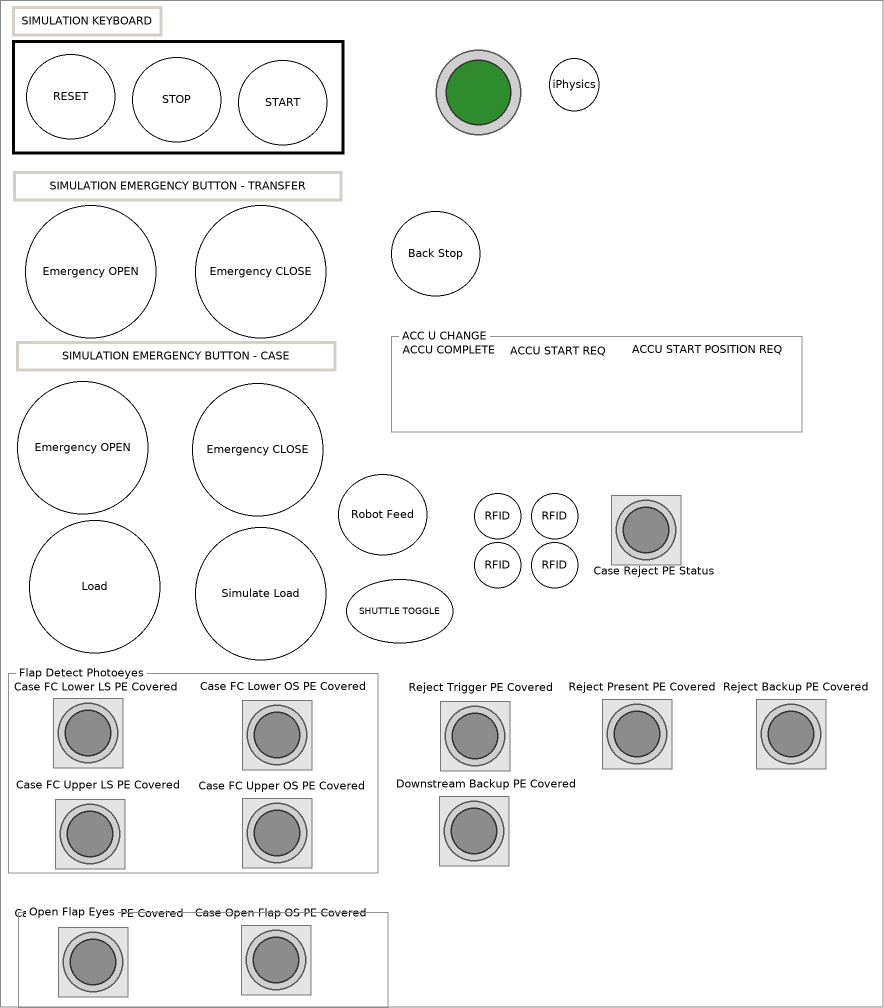
VISUALIZATION Casepacker_Keyboard  // 884x1008
    Rectangle (12,40 332x114)
    Ellipse (26,54 89x85), "RESET"
        tap csp_transfer_main_services_pushbuttons.visu_reset
    Ellipse (132,57 89x85), "STOP"
        tap csp_transfer_main_services_pushbuttons.visu_stop
    Ellipse (238,60 89x85), "START"
        tap csp_transfer_main_services_pushbuttons.visu_start
    Textfield (12,6 150x30), "SIMULATION KEYBOARD"
    Ellipse (25,205 131x133), "Emergency OPEN"
        tap csp_transfer_main_services_pushbuttons.visu_emergency_open
    Ellipse (195,205 131x133), "Emergency CLOSE"
        tap csp_transfer_main_services_pushbuttons.visu_emergency_close
    Textfield (13,171 329x30), "SIMULATION EMERGENCY BUTTON - TRANSFER"
    Lamp1 (426,43 105x99), variable: csp_transfer_main_safety_emergency.HMI_button_lamp_do.field.status, style: Lamp-Lamp1-Green
    Ellipse (391,211 89x85), "Back Stop", colour toggle: csp_transfer_upstacker_sensors.debug_carton_backstop
        toggle csp_transfer_upstacker_sensors.debug_carton_backstop
    Ellipse (192,383 131x133), "Emergency CLOSE"
        tap csp_case_main_services_pushbuttons.visu_emergency_close
    Textfield (16,341 320x30), "SIMULATION EMERGENCY BUTTON - CASE"
    Ellipse (17,381 131x133), "Emergency OPEN"
        tap csp_case_main_services_pushbuttons.visu_emergency_open
    Ellipse (549,58 50x53), "iPhysics"
        toggle MAIN.IP_enable
    GroupBox (8,665 370x208), "Flap Detect Photoeyes"
        PushSwitchLed (45,33 70x70), variable: dbg_csp_case_fc_ls_lower_sensors.flap_chksect_shd.force_input_status, behaviour: TOGGLE, style: Switch-PushSwitchLed-Gray
    Ellipse (29,520 131x133), "Load"
        tap csp_case_loader.load_request
    Ellipse (531,493 47x46), "RFID"
        toggle csp_case_closing_ls_upper.rfid_fake
    Ellipse (531,542 47x46), "RFID"
        toggle csp_case_closing_ls_lower.rfid_fake
    Ellipse (474,493 47x46), "RFID"
        toggle csp_case_closing_os_upper.rfid_fake
    Ellipse (474,542 47x46), "RFID"
        toggle csp_case_closing_os_lower.rfid_fake
    PushSwitchLed (611,495 70x70), behaviour: TOGGLE, style: Switch-PushSwitchLed-Gray
    Label (579,556 150x30), "Case Reject PE Status"
    Ellipse (195,527 131x133), "Simulate Load"
        tap csp_case_transport.product_loaded
    Label (8,673 176x28), "Case FC Lower LS PE Covered"
    PushSwitchLed (55,799 70x70), variable: dbg_csp_case_fc_ls_upper_sensors.flap_chksect_shd.force_input_status, behaviour: TOGGLE, style: Switch-PushSwitchLed-Gray
    Label (10,775 176x20), "Case FC Upper LS PE Covered"
    PushSwitchLed (242,700 70x70), variable: dbg_csp_case_fc_os_lower_sensors.flap_chksect_shd.force_input_status, behaviour: TOGGLE, style: Switch-PushSwitchLed-Gray
    Label (195,678 176x17), "Case FC Lower OS PE Covered"
    PushSwitchLed (242,798 70x70), variable: dbg_csp_case_fc_os_upper_sensors.flap_chksect_shd.force_input_status, behaviour: TOGGLE, style: Switch-PushSwitchLed-Gray
    Label (194,777 176x18), "Case FC Upper OS PE Covered"
    Label (8,888 176x28)
    PushSwitchLed (58,927 70x70), variable: dbg_csp_case_openflap_sensors.open_flap_ls_di_dchk_shd.force_input_status, behaviour: TOGGLE, style: Switch-PushSwitchLed-Gray
    Label (11,905 176x17), "Case Open Flap LS PE Covered"
    PushSwitchLed (241,925 70x70), variable: dbg_csp_case_openflap_sensors.open_flap_os_di_dchk_shd.force_input_status, behaviour: TOGGLE, style: Switch-PushSwitchLed-Gray
    Label (193,904 176x18), "Case Open Flap OS PE Covered"
    GroupBox (391,328 411x104), "ACC U CHANGE"
        Label (381,-232 176x28)
        Label (79,9 176x28), "ACCU START REQ"
    PushSwitchLed (440,701 70x70), variable: dbg_csp_case_discharge_reject_sensors.reject_trigger_inchoerence_chksect_shd.force_input_status, behaviour: TOGGLE, style: Switch-PushSwitchLed-Gray
    Label (393,679 176x17), "Reject Trigger PE Covered"
    PushSwitchLed (602,699 70x70), variable: dbg_csp_case_discharge_reject_sensors.reject_present_di_shd.is_covered, behaviour: TOGGLE, style: Switch-PushSwitchLed-Gray
    Label (554,678 176x18), "Reject Present PE Covered"
    PushSwitchLed (756,699 70x70), variable: dbg_csp_case_discharge_reject_sensors.reject_backup_di_shd.is_covered, behaviour: TOGGLE, style: Switch-PushSwitchLed-Gray
    Label (708,678 176x18), "Reject Backup PE Covered"
    PushSwitchLed (439,796 70x70), variable: dbg_csp_case_discharge_reject_sensors.downstream_backup_di_shd.is_covered, behaviour: TOGGLE, style: Switch-PushSwitchLed-Gray
    Label (391,775 190x18), "Downstream Backup PE Covered"
    Ellipse (338,474 89x81), "Robot Feed"
        toggle csp_case_feed.Feed_request
    Ellipse (346,579 107x64), "SHUTTLE TOGGLE"
        toggle csp_case_transport.product_loaded
    GroupBox (18,904 370x104), "Open Flap Eyes"
        Label (381,-232 176x28)
    Label (361,336 176x28), "ACCU COMPLETE"
    Label (619,327 176x45), "ACCU START POSITION REQ"
END_VISUALIZATION

(* stored: Version 1.1.0.1, ProductVersion 3.1.4024.3
   Visu Casepacker_Keyboard: Id {ba2757c6-980f-4151-a36a-574c751732a5} *)
